FUNCTION_BLOCK SPLIT_MI_DO_S_Octal_SA (* Splits a DataPanel_MI_DO_S_Octal_SA into 8 DataPanel_MI_DO_S_Single_SA *)
  (* Standard: 61499-2; Description: Copyright (c) 2026 HR Agrartechnik GmbH SPDX-License-Identifier: EPL-2.0 *)
  (* Version 1.0, 2026-05-28, franz, HR Agrartechnik GmbH *)
  PACKAGE DataPanel::io::MI::DQ;
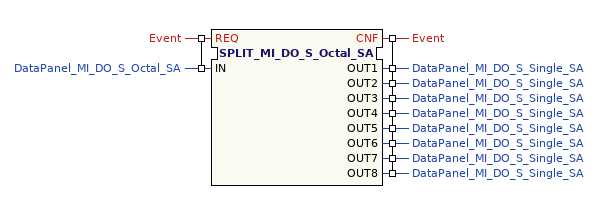
  EVENT_INPUT
    REQ WITH IN; (* Service Request *)
  END_EVENT
  EVENT_OUTPUT
    CNF WITH OUT1, OUT2, OUT3, OUT4, OUT5, OUT6, OUT7, OUT8; (* Confirmation of Requested Service *)
  END_EVENT
  VAR_INPUT
    IN : DataPanel::io::MI::DQ::DataPanel_MI_DO_S_Octal_SA; (* Octal Input *)
  END_VAR
  VAR_OUTPUT
    OUT1 : DataPanel::io::MI::DQ::DataPanel_MI_DO_S_Single_SA; (* Single Output 1 *)
    OUT2 : DataPanel::io::MI::DQ::DataPanel_MI_DO_S_Single_SA; (* Single Output 2 *)
    OUT3 : DataPanel::io::MI::DQ::DataPanel_MI_DO_S_Single_SA; (* Single Output 3 *)
    OUT4 : DataPanel::io::MI::DQ::DataPanel_MI_DO_S_Single_SA; (* Single Output 4 *)
    OUT5 : DataPanel::io::MI::DQ::DataPanel_MI_DO_S_Single_SA; (* Single Output 5 *)
    OUT6 : DataPanel::io::MI::DQ::DataPanel_MI_DO_S_Single_SA; (* Single Output 6 *)
    OUT7 : DataPanel::io::MI::DQ::DataPanel_MI_DO_S_Single_SA; (* Single Output 7 *)
    OUT8 : DataPanel::io::MI::DQ::DataPanel_MI_DO_S_Single_SA; (* Single Output 8 *)
  END_VAR
  EC_STATES
    REQ : REQ -> CNF;
  END_STATES
  ALGORITHM REQ IN ST: (* Normally executed algorithm *)
OUT1.u8SAMember := IN.u8SAMember;
OUT1.Port := IN.Port1;
OUT2.u8SAMember := IN.u8SAMember;
OUT2.Port := IN.Port2;
OUT3.u8SAMember := IN.u8SAMember;
OUT3.Port := IN.Port3;
OUT4.u8SAMember := IN.u8SAMember;
OUT4.Port := IN.Port4;
OUT5.u8SAMember := IN.u8SAMember;
OUT5.Port := IN.Port5;
OUT6.u8SAMember := IN.u8SAMember;
OUT6.Port := IN.Port6;
OUT7.u8SAMember := IN.u8SAMember;
OUT7.Port := IN.Port7;
OUT8.u8SAMember := IN.u8SAMember;
OUT8.Port := IN.Port8;
  END_ALGORITHM
END_FUNCTION_BLOCK
